// TIA Portal V18 export
FUNCTION "CylinderCtrl_V2" : Void   // FC3011, SCL
TITLE = CylinderV3
{ S7_Optimized_Access := 'FALSE' }
AUTHOR : JM
FAMILY : RCS
VERSION : 18.2
// this function is only used for cylinder control
// stored: AutoNumber false, SetENOAutomatically true
   VAR_INPUT
      iReset : Bool;   // reset action
      iRun : Bool;   // system run
      iEStop : Bool;   // e_stop monitor
      iManualMode : Bool;   // manual mode
      iAutoMode : Bool;   // auto mode
      iEnableAlarm : Bool;   // alarm will popup up
      iPulse100mS : Bool;   // pulse *100ms
      iPulse1S : Bool;   // pulse*1s
      iCyDBNO : Word;   // Interface data block number
      iCyCounts : Int;   // total counts of cylinder to be used[must be>=1 and <=100]
      iDevAlarmDBNum : Word;   // Device Alarm DataBlock Alarm
   END_VAR
   VAR_TEMP
      CyInterface : "Cyl";
      CyRany : Any;
      cyRSany AT CyRany : Struct
         SyntaxID : Byte;
         DataType : Byte;
         RepetitionFactor : Int;
         DB_Number : Word;
         MemoryAreaAddress : DWord;
      END_STRUCT;
      CyDany : Any;
      CyDSany AT CyDany : Struct
         SyntaxID : Byte;
         DataType : Byte;
         RepetitionFactor : Int;
         DB_Number : Word;
         MemoryAreaAddress : DWord;
      END_STRUCT;
      tpCounts : Int;
      tpi : Int;
      tpRetVal : Int;
   END_VAR
BEGIN
   //---------------------------------------------------------------//
   //FunctionName:CylinderV3
   //FunctionDescription:Cylinder Control block
   //---------------------------------------------------------------//
   (*in:

   #iReset  Bool            reset action
   #iRun    Bool            system run
   #iE_stop Bool            e_stop monitor
   #iManualMode Bool        manual mode
   #iAutoMode   Bool        auto mode
   #iEnableAlarm    Bool        alarm will popup up
   #iPulse_100mS    Bool        pulse *100ms
   iPulse_1S   Bool        pulse*1s
   iCyDBNO Int Int     Interface data block number
   iCyCounts   Int     total counts OF "Cylinder" TO be used[must be>=1 AND <=100]

   //inout:
   //out:
   *)
   //---------------------------------------------------------------//
   //Version:V3
   //D&T:2016-11-14
   //Group:RCS
   //Author:JiangMing
   //-------------------------Modify1----------------------------------//
   //Version:
   //D&T:2016-11-17
   //Group: RCS
   //Author:JiangMing
   //Modify:Update cylinder no as output interface
   //-------------------------Modify2----------------------------------//
   //Version:       V18.3
   //D&T:           2020-06-11
   //Group:         RCS
   //Author:        JM
   //Modify:        1.MaxCylinder count 200 
   //               2.Refine alarm interface
   IF #iCyCounts > 200 THEN
       #tpCounts := 200;
   ELSE
       #tpCounts := #iCyCounts;
   END_IF;
   //input

   FOR #tpi := 0 TO #tpCounts-1 DO
       //****************************************************************************************//
       #cyRSany.SyntaxID := 16#10;
       #cyRSany.DataType := 16#02;
       #cyRSany.RepetitionFactor := 22;
       #cyRSany.DB_Number := #iCyDBNO;
       #cyRSany.MemoryAreaAddress := 16#8400_0000 OR (SHL(IN := INT_TO_DWORD(#tpi * 22), N := 3));///
       //-----------------------------//
       #CyDSany.SyntaxID := 16#10;
       #CyDSany.DataType := 16#02;
       #CyDSany.RepetitionFactor := 22;
       #CyDSany.DB_Number := 0;
       #CyDSany.MemoryAreaAddress := 16#8700_0000 OR (SHL(IN := INT_TO_DWORD(0), N := 3));///
       #tpRetVal := BLKMOV(SRCBLK := #CyRany, DSTBLK => #CyDany);
       //***************************************************************************************//
       "CylinderModule_V2"(iReset := #iReset,
                        iRun := #iRun,
                        iEStop := #iEStop,
                        iManualMode := #iManualMode,
                        iAutoMode := #iAutoMode,
                        iEnableAlarm := #iEnableAlarm,
                        iPulse100mS := #iPulse100mS,
                        iPulse1S := #iPulse1S,
                        iError := #CyInterface.In.Error,
                        iGoWorkInterlock := #CyInterface.In.GoWorkInterlock,
                        iGoHomeInterlock := #CyInterface.In.GoHomeInterlock,
                        iWorkPositionSensor := #CyInterface.In.WorkPositionSensor,
                        iHomePositionSensor := #CyInterface.In.HomePositionSensor,
                        iValveType := #CyInterface.In.ValveType,
                        iManualOutputType := #CyInterface.In.ManualOutputType,
                        iFaultTime := #CyInterface.In.FaultTime,
                        iOnPositionTime := #CyInterface.In.OnPositionTime,
                           ioResetOut:=#CyInterface.Inout.ResetOut,
                        ioGoWorkPosition := #CyInterface.Out.GoWorkPosition,
                        ioGoHomePosition := #CyInterface.Out.GoHomePosition,
                        oGoWP_ButtonActive => #CyInterface.Out.GoWPButtonActive,
                        oGoHP_ButtonActive => #CyInterface.Out.GoHPButtonActive,
                        ioGoWorkFault := #CyInterface.Out.GoWorkFault,
                        ioGoHomeFault := #CyInterface.Out.GoHomeFault,
                        ioSensorPositionFault := #CyInterface.Out.SensorPositionFault,
                        oCyNo => #CyInterface.Out.CyNO,
                        ioManualGoWork := #CyInterface.Inout.ManualGoWork,
                        ioManualGoHome := #CyInterface.Inout.ManualGoHome,
                        ioAutoGoWork := #CyInterface.Inout.AutoGoWork,
                        ioAutoGoHome := #CyInterface.Inout.AutoGoHome,
                        ioGoWorkTime := #CyInterface.S.GoWorkTime,
                        ioGoHomeTime := #CyInterface.S.GoHomeTime,
                        ioWorkFaultTime := #CyInterface.S.WorkFaultTime,
                        ioHomeFaultTime := #CyInterface.S.HomeFaultTime,
                        ioBothSensorOnTime := #CyInterface.S.BothSensorOnTime,
                        ioPulse100mSP := #CyInterface.S.Pulse100mSP,
                        ioAutoGoWorkP := #CyInterface.S.AutoGoWorkP,
                        ioAutoGoHomeP := #CyInterface.S.AutoGoHomeP,
                        ioGoWork100mSP := #CyInterface.S.GoWork100mSP,
                        ioGoHome100mSP := #CyInterface.S.GoHome100mSP,
                        ioBothSensorOn100mSP := #CyInterface.S.BothSensorOn100mSP,
                        ioAlarm := #CyInterface.S.Alarm,
                        ioSpare1 := #CyInterface.S.spare1,
                        ioSpare2 := #CyInterface.S.spare2);
       //*******************************************************************************//
         POKE_BOOL(area := 16#84,
                   bitOffset := 4 * (#tpi MOD 2) + 0,
                   byteOffset :=  #tpi / 2,
                   dbNumber := #iDevAlarmDBNum,
                   value := #CyInterface.Out.GoWorkFault);
         POKE_BOOL(area := 16#84,
                   bitOffset := 4 * (#tpi MOD 2) + 1,
                   byteOffset :=  #tpi / 2,
                   dbNumber := #iDevAlarmDBNum,
                   value := #CyInterface.Out.GoHomeFault);
         POKE_BOOL(area := 16#84,
                   bitOffset := 4 * (#tpi MOD 2) + 2,
                   byteOffset :=  #tpi / 2,
                   dbNumber := #iDevAlarmDBNum,
                   value := #CyInterface.Out.SensorPositionFault);
       #CyInterface.Out.CyNO := INT_TO_BYTE(#tpi+1);
       //output
       #cyRSany.SyntaxID := 16#10;
       #cyRSany.DataType := 16#02;
       #cyRSany.RepetitionFactor := 16;
       #cyRSany.DB_Number := 0;
       #cyRSany.MemoryAreaAddress := 16#8700_0000 OR (SHL(IN := INT_TO_DWORD(6), N := 3));///
       //-----------------------------//
       #CyDSany.SyntaxID := 16#10;
       #CyDSany.DataType := 16#02;
       #CyDSany.RepetitionFactor := 16;
       #CyDSany.DB_Number := #iCyDBNO;
       #CyDSany.MemoryAreaAddress := 16#8400_0000 OR (SHL(IN := INT_TO_DWORD(#tpi* 22 + 6), N := 3));///
       #tpRetVal := BLKMOV(SRCBLK := #CyRany, DSTBLK => #CyDany);
       //******************************************************************************//


   END_FOR;
END_FUNCTION
